// TIA Portal V15.1 export
// export: Created 2024-06-21T08:41:20.9813268Z, ExportSetting WithDefaults, DisplayName Totally Integrated Automation Portal, DisplayVersion V15.1 Update 5, DisplayName TIA Portal Openness, DisplayVersion V15.1 Update 5, DisplayName SINAMICS Startdrive Advanced, DisplayVersion V15.1, DisplayName G130, G150, S120, S150, SINAMICS MV, S210, DisplayVersion V15.1, DisplayName G110M, G120, G120C, G120D, G120P, DisplayVersion V15.1, DisplayName STEP 7 Professional, DisplayVersion V15.1 Update 5, DisplayName STEP 7 Safety, DisplayVersion V15.1, DisplayName WinCC Professional, DisplayVersion V15.1 Update 5, DisplayName SIMATIC Visualization Architect, DisplayVersion V15.1
FUNCTION_BLOCK "LVIDSMaster"   // FB1201, SCL
TITLE = LVIDSMaster
{ S7_Optimized_Access := 'FALSE' }
VERSION : 0.1
// stored: AutoNumber false, IsIECCheckEnabled false, SetENOAutomatically False, UDAEnableTagReadback false
   VAR_INPUT
      C_SubSystem { ExternalAccessible := 'False'; ExternalVisible := 'False'; ExternalWritable := 'False'} : Int;   // VDComm - Subsystem
      C_VDCommMasterRcvDB { ExternalAccessible := 'False'; ExternalVisible := 'False'; ExternalWritable := 'False'} : DB_ANY;   // VDComm - Master receive DB
      C_VDCommMasterSndDB { ExternalAccessible := 'False'; ExternalVisible := 'False'; ExternalWritable := 'False'} : DB_ANY;   // VDComm - Master send DB
      C_VDCommLocalRcvDB { ExternalAccessible := 'False'; ExternalVisible := 'False'; ExternalWritable := 'False'} : DB_ANY;   // VDComm - Local receive DB
      C_VDCommLocalSndDB { ExternalAccessible := 'False'; ExternalVisible := 'False'; ExternalWritable := 'False'} : DB_ANY;   // VDComm - Local send DB
      C_Plant { ExternalAccessible := 'False'; ExternalVisible := 'False'; ExternalWritable := 'False'} : Int;   // Plant ( VCG : 321, VCT : 461, VCCD : 861, VCQD : 862, VCLQ : 863, VCCH : 11 )
      C_IDType { ExternalAccessible := 'False'; ExternalVisible := 'False'; ExternalWritable := 'False'} : DWord;   // Identifier type (0 : Body tag, > 0 : Carrier tag Ex.: Carrier A-shop 162)
      I_OutOfUse { ExternalAccessible := 'False'; ExternalVisible := 'False'; ExternalWritable := 'False'} : Bool;   // Put out of use
      I_PartPres { ExternalAccessible := 'False'; ExternalVisible := 'False'; ExternalWritable := 'False'} : Bool;   // Cycle of tag data use active / Part is present in station
      I_TagID { ExternalAccessible := 'False'; ExternalVisible := 'False'; ExternalWritable := 'False'} : DWord;   // Tag identification ( to get VEM data )
      I_BodyID { ExternalAccessible := 'False'; ExternalVisible := 'False'; ExternalWritable := 'False'} : DWord;   // Body identification ( to get VEM data )
      I_CarrierID { ExternalAccessible := 'False'; ExternalVisible := 'False'; ExternalWritable := 'False'} : DWord;   // Carrier identification ( to get VEM data )
      I_MixNbr { ExternalAccessible := 'False'; ExternalVisible := 'False'; ExternalWritable := 'False'} : DWord;   // Mixnumber ( to get VEM data )
      I_PopID { ExternalAccessible := 'False'; ExternalVisible := 'False'; ExternalWritable := 'False'} : UDInt;   // Spare Data / PopID ( to get VEM data )
      I_PopIDSuffix { ExternalAccessible := 'False'; ExternalVisible := 'False'; ExternalWritable := 'False'} : Char;   // PopID suffix ( to get VEM data )
      I_PopType { ExternalAccessible := 'False'; ExternalVisible := 'False'; ExternalWritable := 'False'} : UDInt;   // Pop identifier ( to get VEM data )
      I_StartGetVEMData { ExternalAccessible := 'False'; ExternalVisible := 'False'; ExternalWritable := 'False'} : Bool;   // Get VEM data - Start on edge
      I_ResetAlarm { ExternalAccessible := 'False'; ExternalVisible := 'False'; ExternalWritable := 'False'} : Bool;   // Reset alarm
   END_VAR
   VAR_OUTPUT
      O_VEMDataValid { ExternalAccessible := 'False'; ExternalVisible := 'False'; ExternalWritable := 'False'} : Bool;   // VEM data is valid
      O_VEMDataNotValid { ExternalAccessible := 'False'; ExternalVisible := 'False'; ExternalWritable := 'False'} : Bool;   // VEM data is not valid
      O_GetVEMDataBusy { ExternalAccessible := 'False'; ExternalVisible := 'False'; ExternalWritable := 'False'} : Bool;   // Get VEM data - Busy
      O_Status { ExternalAccessible := 'False'; ExternalVisible := 'False'; ExternalWritable := 'False'} : Int;   // 0: no activity, 1: OK-Data valid, 2: Busy, -1..-32768: error code / 0: no activity, 1: OK-Get VEM data valid, 2: Busy, -1..-32768: error code
      O_Alarm { ExternalAccessible := 'False'; ExternalVisible := 'False'; ExternalWritable := 'False'} : Bool;   // Get VEM Data Alarm (Status < 0)
   END_VAR
   VAR_IN_OUT
      IO_VDComm : "VDComm";   // VD Comm / VD Comm - communication record
      IO_VIDS : "VIDS";   // VIDS - internal record
      IO_VEMData : "VEMData";   // VEM data - received
      IO_VEMDataChange : "VEMData";   // VEM data - to be changed
      IO_SpecificData : Array[0..7925] of Byte;   // Specific data received
      IO_Alarm : "Alarm";   // Alarm
      H_Master : "H_LVIDSMaster";   // Animation
      H_HMI : "H_HMI";   // Used for icon animation
   END_VAR
   VAR DB_SPECIFIC
      i { ExternalAccessible := 'False'; ExternalVisible := 'False'; ExternalWritable := 'False'} : Int;   // Index
      PartPres { ExternalAccessible := 'False'; ExternalVisible := 'False'; ExternalWritable := 'False'} : Bool;
      PartLostDlyTmrElapsed { ExternalAccessible := 'False'; ExternalVisible := 'False'; ExternalWritable := 'False'} : Bool;
      PartLostDlyTmrAct { ExternalAccessible := 'False'; ExternalVisible := 'False'; ExternalWritable := 'False'} : DInt;
      VEMDataChangeIoSerial { ExternalAccessible := 'False'; ExternalVisible := 'False'; ExternalWritable := 'False'} : Bool;
      VEMDataChangeHMISerial { ExternalAccessible := 'False'; ExternalVisible := 'False'; ExternalWritable := 'False'} : Array[0..255] of Byte;
      VEMDataChangeHMI { ExternalAccessible := 'False'; ExternalVisible := 'False'; ExternalWritable := 'False'; S7_SetPoint := 'True'} : "VEMData";
      VEMDataInitArray { ExternalAccessible := 'False'; ExternalVisible := 'False'; ExternalWritable := 'False'} : Array[0..255] of Byte;   // VEM data in serialized form
      VEMDataRcvArray { ExternalAccessible := 'False'; ExternalVisible := 'False'; ExternalWritable := 'False'} : Array[0..255] of Byte;   // VEM data in serialized form
      VEMDataRcv { ExternalAccessible := 'False'; ExternalVisible := 'False'; ExternalWritable := 'False'; S7_SetPoint := 'True'} : "VEMData";
      VEMDataSndArray { ExternalAccessible := 'False'; ExternalVisible := 'False'; ExternalWritable := 'False'} : Array[0..255] of Byte;
      SpecificData { ExternalAccessible := 'False'; ExternalVisible := 'False'; ExternalWritable := 'False'} : Array[0..7925] of Byte;
      VEMDataValid { ExternalAccessible := 'False'; ExternalVisible := 'False'; ExternalWritable := 'False'} : Bool;
      VEMDataNotValid { ExternalAccessible := 'False'; ExternalVisible := 'False'; ExternalWritable := 'False'} : Bool;
      CmdCodeSent { ExternalAccessible := 'False'; ExternalVisible := 'False'; ExternalWritable := 'False'} : DWord;   // Command code sent to VD
      CmdCodeRcvd { ExternalAccessible := 'False'; ExternalVisible := 'False'; ExternalWritable := 'False'} : DWord;   // Command code received from VD
      TagIDMem { ExternalAccessible := 'False'; ExternalVisible := 'False'; ExternalWritable := 'False'} : DWord;
      BodyIDMem { ExternalAccessible := 'False'; ExternalVisible := 'False'; ExternalWritable := 'False'} : DWord;
      CarrierIDMem { ExternalAccessible := 'False'; ExternalVisible := 'False'; ExternalWritable := 'False'} : DWord;
      MixNbrMem { ExternalAccessible := 'False'; ExternalVisible := 'False'; ExternalWritable := 'False'} : DWord;
      PopIDMem { ExternalAccessible := 'False'; ExternalVisible := 'False'; ExternalWritable := 'False'} : UDInt;   // Spare Data / PopID
      PopIDSuffixMem { ExternalAccessible := 'False'; ExternalVisible := 'False'; ExternalWritable := 'False'} : Char;   // PopID suffix
      PopTypeMem { ExternalAccessible := 'False'; ExternalVisible := 'False'; ExternalWritable := 'False'} : UDInt;   // Spare Data / Pop Identifier
      CarTypeVariant { ExternalAccessible := 'False'; ExternalVisible := 'False'; ExternalWritable := 'False'} : Int;   // Car type - Decoded from variant
      CarTypeBody { ExternalAccessible := 'False'; ExternalVisible := 'False'; ExternalWritable := 'False'} : Int;   // Car type - Decoded from bodytype matrix
      SteeringVariant { ExternalAccessible := 'False'; ExternalVisible := 'False'; ExternalWritable := 'False'} : Int;
      SteeringBody { ExternalAccessible := 'False'; ExternalVisible := 'False'; ExternalWritable := 'False'} : Int;
      CarTypeArray { ExternalAccessible := 'False'; ExternalVisible := 'False'; ExternalWritable := 'False'} : Array[1..3] of Int;
      DataValidSnd { ExternalAccessible := 'False'; ExternalVisible := 'False'; ExternalWritable := 'False'} : Bool;   // Data valid - Send
      DataRcvOk { ExternalAccessible := 'False'; ExternalVisible := 'False'; ExternalWritable := 'False'} : Bool;
      DataRcvNok { ExternalAccessible := 'False'; ExternalVisible := 'False'; ExternalWritable := 'False'} : Bool;
      DeserializePos { ExternalAccessible := 'False'; ExternalVisible := 'False'; ExternalWritable := 'False'} : DInt;
      SerializePos { ExternalAccessible := 'False'; ExternalVisible := 'False'; ExternalWritable := 'False'} : DInt;
      SequenceTotalOvertime { ExternalAccessible := 'False'; ExternalVisible := 'False'; ExternalWritable := 'False'} : Time;
      StartChangeVEMDataEdg { ExternalAccessible := 'False'; ExternalVisible := 'False'; ExternalWritable := 'False'} : Bool;   // Change VEM data - Start edge
      StartChangeVEMDataPls { ExternalAccessible := 'False'; ExternalVisible := 'False'; ExternalWritable := 'False'} : Bool;   // Change VEM data - Start pulse
      SeqOvTimeElapsed { ExternalAccessible := 'False'; ExternalVisible := 'False'; ExternalWritable := 'False'} : Bool;
      CodeBusy { ExternalAccessible := 'False'; ExternalVisible := 'False'; ExternalWritable := 'False'} : Int;
      RetVal { ExternalAccessible := 'False'; ExternalVisible := 'False'; ExternalWritable := 'False'} : Int;   // Return value
      GetVEMDataByRFIDBeginReqEdg { ExternalAccessible := 'False'; ExternalVisible := 'False'; ExternalWritable := 'False'} : Bool;
      GetVEMDataByTagReplBeginReqEdg { ExternalAccessible := 'False'; ExternalVisible := 'False'; ExternalWritable := 'False'} : Bool;
      DataValidRcvGetVEMDataByRFID { ExternalAccessible := 'False'; ExternalVisible := 'False'; ExternalWritable := 'False'} : Bool;
      GetVEMDataBeginReqEdg { ExternalAccessible := 'False'; ExternalVisible := 'False'; ExternalWritable := 'False'} : Bool;
      GetVEMDataByHMIBeginEdg { ExternalAccessible := 'False'; ExternalVisible := 'False'; ExternalWritable := 'False'} : Bool;
      GetVEMDataRcvOk { ExternalAccessible := 'False'; ExternalVisible := 'False'; ExternalWritable := 'False'} : Bool;
      ChangeDataReq { ExternalAccessible := 'False'; ExternalVisible := 'False'; ExternalWritable := 'False'} : Bool;
      ChangeDataReqEdg { ExternalAccessible := 'False'; ExternalVisible := 'False'; ExternalWritable := 'False'} : Bool;
      ChangeDataBeginReqEdg { ExternalAccessible := 'False'; ExternalVisible := 'False'; ExternalWritable := 'False'} : Bool;
      ChangeDataRcvOk { ExternalAccessible := 'False'; ExternalVisible := 'False'; ExternalWritable := 'False'} : Bool;
      GetNextIDBeginReqEdg { ExternalAccessible := 'False'; ExternalVisible := 'False'; ExternalWritable := 'False'} : Bool;
      GetNextIDRcvOk { ExternalAccessible := 'False'; ExternalVisible := 'False'; ExternalWritable := 'False'} : Bool;
      ReplaceTagReq { ExternalAccessible := 'False'; ExternalVisible := 'False'; ExternalWritable := 'False'} : Bool;
      ReplaceTagReqEdg { ExternalAccessible := 'False'; ExternalVisible := 'False'; ExternalWritable := 'False'} : Bool;
      ReplaceTagBeginReqEdg { ExternalAccessible := 'False'; ExternalVisible := 'False'; ExternalWritable := 'False'} : Bool;
      ReplaceTagRcvOk { ExternalAccessible := 'False'; ExternalVisible := 'False'; ExternalWritable := 'False'} : Bool;
      InitTagBeginReqEdg { ExternalAccessible := 'False'; ExternalVisible := 'False'; ExternalWritable := 'False'} : Bool;
      InitTagRcvOk { ExternalAccessible := 'False'; ExternalVisible := 'False'; ExternalWritable := 'False'} : Bool;
      GetSpecDataReq { ExternalAccessible := 'False'; ExternalVisible := 'False'; ExternalWritable := 'False'} : Bool;
      GetSpecDataReqEdg { ExternalAccessible := 'False'; ExternalVisible := 'False'; ExternalWritable := 'False'} : Bool;
      GetSpecDataBeginReqEdg { ExternalAccessible := 'False'; ExternalVisible := 'False'; ExternalWritable := 'False'} : Bool;
      GetSpecDataRcvOk { ExternalAccessible := 'False'; ExternalVisible := 'False'; ExternalWritable := 'False'} : Bool;
      PutSpecDataBeginReqEdg { ExternalAccessible := 'False'; ExternalVisible := 'False'; ExternalWritable := 'False'} : Bool;
      PutSpecDataRcvOk { ExternalAccessible := 'False'; ExternalVisible := 'False'; ExternalWritable := 'False'} : Bool;
      TrackBeginReqEdg { ExternalAccessible := 'False'; ExternalVisible := 'False'; ExternalWritable := 'False'} : Bool;   // Tracking - Begin request edge
      TrackingRcvOk { ExternalAccessible := 'False'; ExternalVisible := 'False'; ExternalWritable := 'False'} : Bool;
      CoupleBeginReqEdg { ExternalAccessible := 'False'; ExternalVisible := 'False'; ExternalWritable := 'False'} : Bool;
      CoupleRcvOk { ExternalAccessible := 'False'; ExternalVisible := 'False'; ExternalWritable := 'False'} : Bool;
      DecoupleBeginReqEdg { ExternalAccessible := 'False'; ExternalVisible := 'False'; ExternalWritable := 'False'} : Bool;
      DecoupleRcvOk { ExternalAccessible := 'False'; ExternalVisible := 'False'; ExternalWritable := 'False'} : Bool;
      ConfirmBeginReqEdg { ExternalAccessible := 'False'; ExternalVisible := 'False'; ExternalWritable := 'False'} : Bool;
      ConfirmationRcvOk { ExternalAccessible := 'False'; ExternalVisible := 'False'; ExternalWritable := 'False'} : Bool;
      NoFunctionBusy { ExternalAccessible := 'False'; ExternalVisible := 'False'; ExternalWritable := 'False'} : Bool;
      Busy { ExternalAccessible := 'False'; ExternalVisible := 'False'; ExternalWritable := 'False'} : Bool;
      BtnGetVEMTagIDEdge { ExternalAccessible := 'False'; ExternalVisible := 'False'; ExternalWritable := 'False'} : Bool;
      btnGetVEMDataByMixNbrEdg { ExternalAccessible := 'False'; ExternalVisible := 'False'; ExternalWritable := 'False'} : Bool;
      BtnGetVEMCarrierEdge { ExternalAccessible := 'False'; ExternalVisible := 'False'; ExternalWritable := 'False'} : Bool;
      ChangeDataNotValid { ExternalAccessible := 'False'; ExternalVisible := 'False'; ExternalWritable := 'False'} : Bool;
      MessageLength { ExternalAccessible := 'False'; ExternalVisible := 'False'; ExternalWritable := 'False'} : Word;   // Message Length
      SendToVD { ExternalAccessible := 'False'; ExternalVisible := 'False'; ExternalWritable := 'False'} : Bool;   // Send To PCS
      SendFinished { ExternalAccessible := 'False'; ExternalVisible := 'False'; ExternalWritable := 'False'} : Bool;   // Send Finished / Send data Finished
      RcvOkGetVEMDataCode { ExternalAccessible := 'False'; ExternalVisible := 'False'; ExternalWritable := 'False'} : Bool;
      RcvOkIdentification { ExternalAccessible := 'False'; ExternalVisible := 'False'; ExternalWritable := 'False'} : Bool;
      NewData { ExternalAccessible := 'False'; ExternalVisible := 'False'; ExternalWritable := 'False'} : Bool;   // New Data Is Present
      ResetNewData { ExternalAccessible := 'False'; ExternalVisible := 'False'; ExternalWritable := 'False'} : Bool;   // Reset Data Recevied
      CarrierIDDataReqOk { ExternalAccessible := 'False'; ExternalVisible := 'False'; ExternalWritable := 'False'} : Bool;
      ReqSendReport { ExternalAccessible := 'False'; ExternalVisible := 'False'; ExternalWritable := 'False'} : Bool;
      SendCmd { ExternalAccessible := 'False'; ExternalVisible := 'False'; ExternalWritable := 'False'} : Bool;   // External command send
      ResetAllRequests { ExternalAccessible := 'False'; ExternalVisible := 'False'; ExternalWritable := 'False'} : Bool;
      HMIGetVEMDataTagIDMem { ExternalAccessible := 'False'; ExternalVisible := 'False'; ExternalWritable := 'False'} : DInt;
      HMIGetVEMDataMixNbrMem { ExternalAccessible := 'False'; ExternalVisible := 'False'; ExternalWritable := 'False'} : DInt;
      HMIGetVEMDataCarrIdMem { ExternalAccessible := 'False'; ExternalVisible := 'False'; ExternalWritable := 'False'} : DInt;
      StartGetVEMDataEdg { ExternalAccessible := 'False'; ExternalVisible := 'False'; ExternalWritable := 'False'} : Bool;
      StartGetVEMDataPls { ExternalAccessible := 'False'; ExternalVisible := 'False'; ExternalWritable := 'False'} : Bool;
      Status { ExternalAccessible := 'False'; ExternalVisible := 'False'; ExternalWritable := 'False'} : Int;
      StatusMem { ExternalAccessible := 'False'; ExternalVisible := 'False'; ExternalWritable := 'False'} : Int;
      StepNbr { ExternalAccessible := 'False'; ExternalVisible := 'False'; ExternalWritable := 'False'} : Int;   // Active stepnumber
      Step0ExitPls { ExternalAccessible := 'False'; ExternalVisible := 'False'; ExternalWritable := 'False'} : Bool;   // Step 0 - Pulse created on exit
      Step50EntryEdg { ExternalAccessible := 'False'; ExternalVisible := 'False'; ExternalWritable := 'False'} : Bool;   // Step 50 - Edge created on entry
      Step50EntryPls { ExternalAccessible := 'False'; ExternalVisible := 'False'; ExternalWritable := 'False'} : Bool;   // Step 50 - Pulse created on entry
      Step50ExitEdg { ExternalAccessible := 'False'; ExternalVisible := 'False'; ExternalWritable := 'False'} : Bool;   // Step 50 - Edge created on exit
      Step50ExitPls { ExternalAccessible := 'False'; ExternalVisible := 'False'; ExternalWritable := 'False'} : Bool;   // Step 50 - Pulse created on exit
      Step100EntryEdg { ExternalAccessible := 'False'; ExternalVisible := 'False'; ExternalWritable := 'False'} : Bool;   // Step 100 - Edge created on entry
      Step100EntryPls { ExternalAccessible := 'False'; ExternalVisible := 'False'; ExternalWritable := 'False'} : Bool;   // Step 100 - Pulse created on entry
      Step100ExitEdg { ExternalAccessible := 'False'; ExternalVisible := 'False'; ExternalWritable := 'False'} : Bool;   // Step 100 - Edge created on exit
      Step100ExitPls { ExternalAccessible := 'False'; ExternalVisible := 'False'; ExternalWritable := 'False'} : Bool;   // Step 100 - Pulse created on exit
      Step200EntryEdg { ExternalAccessible := 'False'; ExternalVisible := 'False'; ExternalWritable := 'False'} : Bool;   // Step 200 - Edge created on entry
      Step200EntryPls { ExternalAccessible := 'False'; ExternalVisible := 'False'; ExternalWritable := 'False'} : Bool;   // Step 200 - Pulse created on entry
      Step200ExitEdg { ExternalAccessible := 'False'; ExternalVisible := 'False'; ExternalWritable := 'False'} : Bool;   // Step 200 - Edge created on exit
      Step200ExitPls { ExternalAccessible := 'False'; ExternalVisible := 'False'; ExternalWritable := 'False'} : Bool;   // Step 200 - Pulse created on exit
      Step300EntryEdg { ExternalAccessible := 'False'; ExternalVisible := 'False'; ExternalWritable := 'False'} : Bool;   // Step 300 - Edge created on entry
      Step300EntryPls { ExternalAccessible := 'False'; ExternalVisible := 'False'; ExternalWritable := 'False'} : Bool;   // Step 300 - Pulse created on entry
      Step300ExitEdg { ExternalAccessible := 'False'; ExternalVisible := 'False'; ExternalWritable := 'False'} : Bool;   // Step 300 - Edge created on exit
      Step300ExitPls { ExternalAccessible := 'False'; ExternalVisible := 'False'; ExternalWritable := 'False'} : Bool;   // Step 300 - Pulse created on exit
      Step400ExitEdg { ExternalAccessible := 'False'; ExternalVisible := 'False'; ExternalWritable := 'False'} : Bool;   // Step 400 - Edge created on exit
      Step400ExitPls { ExternalAccessible := 'False'; ExternalVisible := 'False'; ExternalWritable := 'False'} : Bool;   // Step 400 - Pulse created on exit
      Step0To50Cond { ExternalAccessible := 'False'; ExternalVisible := 'False'; ExternalWritable := 'False'} : Bool;   // Step 0 to 50 - Condition
      Step50To100Cond { ExternalAccessible := 'False'; ExternalVisible := 'False'; ExternalWritable := 'False'} : Bool;   // Step 0 to 100 - Condition
      Step50To200Cond { ExternalAccessible := 'False'; ExternalVisible := 'False'; ExternalWritable := 'False'} : Bool;   // Step 0 to 200 - Condition
      Step100To300Cond1 { ExternalAccessible := 'False'; ExternalVisible := 'False'; ExternalWritable := 'False'} : Bool;   // Step 100 to 300 - Condition 1
      Step100To300Cond2 { ExternalAccessible := 'False'; ExternalVisible := 'False'; ExternalWritable := 'False'} : Bool;   // Step 100 to 300 - Condition 2
      Step100To300Cond { ExternalAccessible := 'False'; ExternalVisible := 'False'; ExternalWritable := 'False'} : Bool;   // Step 100 to 300 - Condition
      Step200To300Cond { ExternalAccessible := 'False'; ExternalVisible := 'False'; ExternalWritable := 'False'} : Bool;   // Step 200 to 300 - Condition
      Step300To400Cond { ExternalAccessible := 'False'; ExternalVisible := 'False'; ExternalWritable := 'False'} : Bool;   // Step 300 to 400 - Condition
      Step300To400Cond1 { ExternalAccessible := 'False'; ExternalVisible := 'False'; ExternalWritable := 'False'} : Bool;   // Step 300 to 400 - Condition 1
      Step300To400Cond2 { ExternalAccessible := 'False'; ExternalVisible := 'False'; ExternalWritable := 'False'} : Bool;   // Step 300 to 400 - Condition 2
      Step400To0Cond { ExternalAccessible := 'False'; ExternalVisible := 'False'; ExternalWritable := 'False'} : Bool;   // Step 400 to 0 - Condition
      DataRcvOkGetSpecData { ExternalAccessible := 'False'; ExternalVisible := 'False'; ExternalWritable := 'False'} : Bool;
      VEMDataRcvOKCond1 { ExternalAccessible := 'False'; ExternalVisible := 'False'; ExternalWritable := 'False'} : Bool;
      VEMDataRcvOKCond2 { ExternalAccessible := 'False'; ExternalVisible := 'False'; ExternalWritable := 'False'} : Bool;
      VDCommLocalSndDB { ExternalAccessible := 'False'; ExternalVisible := 'False'; ExternalWritable := 'False'} : Int;   // Send DB / VD Comm - Local send DB number
      VDCommLocalRcvDB { ExternalAccessible := 'False'; ExternalVisible := 'False'; ExternalWritable := 'False'} : Int;   // Recv DB / VD Comm - Local receive DB number
      VD_Identification { ExternalAccessible := 'False'; ExternalVisible := 'False'; ExternalWritable := 'False'} : DWord;   // Identification from VD
      SpecDataLength_DW { ExternalAccessible := 'False'; ExternalVisible := 'False'; ExternalWritable := 'False'} : DWord;
      SpecDataLength_DInt { ExternalAccessible := 'False'; ExternalVisible := 'False'; ExternalWritable := 'False'} : DInt;
      TotalDataSentLength { ExternalAccessible := 'False'; ExternalVisible := 'False'; ExternalWritable := 'False'} : DInt;
      Cmd { ExternalAccessible := 'False'; ExternalVisible := 'False'; ExternalWritable := 'False'} : DWord;
      SeqOvTime { ExternalAccessible := 'False'; ExternalVisible := 'False'; ExternalWritable := 'False'} : Bool;
      OkBegin { ExternalAccessible := 'False'; ExternalVisible := 'False'; ExternalWritable := 'False'} : Bool;
      Step50TmrElapsed { ExternalAccessible := 'False'; ExternalVisible := 'False'; ExternalWritable := 'False'} : Bool;   // Step 50 - Step time elapsed
      Step50TmrAct { ExternalAccessible := 'False'; ExternalVisible := 'False'; ExternalWritable := 'False'} : DInt;   // Step 50 - Step time actual
      Step50TmrActMax { ExternalAccessible := 'False'; ExternalVisible := 'False'; ExternalWritable := 'False'} : DInt;   // Step 50 - Step time actual maximum
      Step100TmrElapsed { ExternalAccessible := 'False'; ExternalVisible := 'False'; ExternalWritable := 'False'} : Bool;   // Step 100 - Step time elapsed
      Step100TmrAct { ExternalAccessible := 'False'; ExternalVisible := 'False'; ExternalWritable := 'False'} : DInt;   // Step 100 - Step time actual
      Step100TmrActMax { ExternalAccessible := 'False'; ExternalVisible := 'False'; ExternalWritable := 'False'} : DInt;   // Step 100 - Step time actual maximum
      Step200TmrElapsed { ExternalAccessible := 'False'; ExternalVisible := 'False'; ExternalWritable := 'False'} : Bool;   // Step 200 - Step time elapsed
      Step200TmrAct { ExternalAccessible := 'False'; ExternalVisible := 'False'; ExternalWritable := 'False'} : DInt;   // Step 200 - Step time actual
      Step200TmrActMax { ExternalAccessible := 'False'; ExternalVisible := 'False'; ExternalWritable := 'False'} : DInt;   // Step 200 - Step time actual maximum
      Step300TmrElapsed { ExternalAccessible := 'False'; ExternalVisible := 'False'; ExternalWritable := 'False'} : Bool;   // Step 300 - Step time elapsed
      Step300TmrAct { ExternalAccessible := 'False'; ExternalVisible := 'False'; ExternalWritable := 'False'} : DInt;   // Step 300 - Step time actual
      Step300TmrActMax { ExternalAccessible := 'False'; ExternalVisible := 'False'; ExternalWritable := 'False'} : DInt;   // Step 300 - Step time actual maximum
      Step400TmrElapsed { ExternalAccessible := 'False'; ExternalVisible := 'False'; ExternalWritable := 'False'} : Bool;   // Step 400 - Step time elapsed
      Step400TmrAct { ExternalAccessible := 'False'; ExternalVisible := 'False'; ExternalWritable := 'False'} : DInt;   // Step 400 - Step time actual
      Step400TmrActMax { ExternalAccessible := 'False'; ExternalVisible := 'False'; ExternalWritable := 'False'} : DInt;   // Step 400 - Step time actual maximum
      EmptyByte { ExternalAccessible := 'False'; ExternalVisible := 'False'; ExternalWritable := 'False'} : Byte;
      PartLostEdg { ExternalAccessible := 'False'; ExternalVisible := 'False'; ExternalWritable := 'False'} : Bool;   // Part lost edge
      PartLostPls { ExternalAccessible := 'False'; ExternalVisible := 'False'; ExternalWritable := 'False'} : Bool;   // Part lost pulse
      PutVemDataTotalLength { ExternalAccessible := 'False'; ExternalVisible := 'False'; ExternalWritable := 'False'} : DInt;
      DataValidRcv { ExternalAccessible := 'False'; ExternalVisible := 'False'; ExternalWritable := 'False'} : Bool;
      BusyGetVEMData { ExternalAccessible := 'False'; ExternalVisible := 'False'; ExternalWritable := 'False'} : Bool;
      Alarm { ExternalAccessible := 'False'; ExternalVisible := 'False'; ExternalWritable := 'False'} : Bool;   // Alarm
      msgPartPresVisible { ExternalAccessible := 'False'; ExternalVisible := 'False'; ExternalWritable := 'False'} : Word;   // HMI - Message animation - Part present - Visible
      msgPartPresAnim { ExternalAccessible := 'False'; ExternalVisible := 'False'; ExternalWritable := 'False'} : Word;   // HMI - Message animation - Part present - Summary
      msgPartNotPresVisible { ExternalAccessible := 'False'; ExternalVisible := 'False'; ExternalWritable := 'False'} : Word;   // HMI - Message animation - Part not present - Visible
      msgPartNotPresAnim { ExternalAccessible := 'False'; ExternalVisible := 'False'; ExternalWritable := 'False'} : Word;   // HMI - Message animation - Part not present - Summary
      IconColour { ExternalAccessible := 'False'; ExternalVisible := 'False'; ExternalWritable := 'False'} : Word;   // Icon colour
      SPACE { ExternalAccessible := 'False'; ExternalVisible := 'False'; ExternalWritable := 'False'} : Char := ' ';
   END_VAR
   VAR
      _Step50Tmr { ExternalAccessible := 'False'; ExternalVisible := 'False'; ExternalWritable := 'False'; S7_SetPoint := 'True'} : "LTimer";   // Step 50 - Timer
      _Step100Tmr { ExternalAccessible := 'False'; ExternalVisible := 'False'; ExternalWritable := 'False'; S7_SetPoint := 'True'} : "LTimer";   // Step 100 - Timer
      _Step200Tmr { ExternalAccessible := 'False'; ExternalVisible := 'False'; ExternalWritable := 'False'; S7_SetPoint := 'True'} : "LTimer";   // Step 200 - Timer
      _Step300Tmr { ExternalAccessible := 'False'; ExternalVisible := 'False'; ExternalWritable := 'False'; S7_SetPoint := 'True'} : "LTimer";   // Step 300 - Timer
      "_LVDComSubSystemS7-1500" { ExternalAccessible := 'False'; ExternalVisible := 'False'; ExternalWritable := 'False'; S7_SetPoint := 'True'} : "LVDComSubSystemS7-1500";
      _PartLostDlyTmr { ExternalAccessible := 'False'; ExternalVisible := 'False'; ExternalWritable := 'False'; S7_SetPoint := 'True'} : "LTimer";   // Part present lost delay timer
   END_VAR
   VAR_TEMP
      ptrIO_VEMData : Any;   // Pointer to received VEM data / Pointer to IO_VEM data
      ptrIO_VEMDataStruct AT ptrIO_VEMData : Struct   // Pointer to IO_VEM data - Structure
         ID : Byte;
         DataType : Byte;
         ReplicationFactor : Word;
         DbNbr : Word;
         CrossAreaPointer : DWord;
      END_STRUCT;
      ptrIO_VEMDataChange : Any;   // Pointer to received VEM data / Pointer to IO_VEM data Change
      ptrIO_VEMDataChangeStruct AT ptrIO_VEMDataChange : Struct   // Pointer to IO_VEM data Change - Structure
         ID : Byte;
         DataType : Byte;
         ReplicationFactor : Word;
         DbNbr : Word;
         CrossAreaPointer : DWord;
      END_STRUCT;
      ptrIO_SpecData : Any;   // Pointer to received VEM data / Pointer to IO_Specific data
      ptrIO_SpecDataStruct AT ptrIO_SpecData : Struct   // Pointer to IO_Specific data - Structure
         ID : Byte;
         DataType : Byte;
         ReplicationFactor : Word;
         DbNbr : Word;
         CrossAreaPointer : DWord;
      END_STRUCT;
      ptrVEMDataVDCommLocalRcv : Any;   // Pointer to received VEM data / Pointer to VEM data in VD local receive DB
      ptrVEMDataVDCommLocalRcvStruct AT ptrVEMDataVDCommLocalRcv : Struct   // Pointer to VEM data in VD local receive DB - Structure
         ID : Byte;
         DataType : Byte;
         ReplicationFactor : Word;
         DbNbr : Word;
         CrossAreaPointer : DWord;
      END_STRUCT;
      ptrVEMDataVDCommLocalSnd : Any;   // Pointer to VEM and specific data to be sent / Pointer to VEM data in VD local send DB
      ptrVEMDataVDCommLocalSndStruct AT ptrVEMDataVDCommLocalSnd : Struct   // Pointer to VEM data in VD local send DB - Structure
         ID : Byte;
         DataType : Byte;
         ReplicationFactor : Word;
         DbNbr : Word;
         CrossAreaPointer : DWord;
      END_STRUCT;
      ptrSpecDataVDCommLocalRcv : Any;   // Pointer to received specific data / Pointer to Specific data in VD local receive DB
      ptrSpecDataVDCommLocalRcvStruct AT ptrSpecDataVDCommLocalRcv : Struct   // Pointer to Specific data in VD local receive DB - Structure
         ID : Byte;
         DataType : Byte;
         ReplicationFactor : Word;
         DbNbr : Word;
         CrossAreaPointer : DWord;
      END_STRUCT;
      ptrSpecDataVDCommLocalSnd : Any;   // Pointer to VEM and specific data to be sent / Pointer to Specific data in VD local send DB
      ptrSpecDataVDCommLocalSndStruct AT ptrSpecDataVDCommLocalSnd : Struct   // Pointer to Specific data in VD local send DB - Structure
         ID : Byte;
         DataType : Byte;
         ReplicationFactor : Word;
         DbNbr : Word;
         CrossAreaPointer : DWord;
      END_STRUCT;
   END_VAR
   VAR CONSTANT
      SECTION_OUTPUTS : Bool := TRUE;   // Section - Outputs
      SECTION_HMI : Bool := TRUE;   // Section - HMI
      PART_LOST_DLY : DInt := 1000;
      VEM_DATA_OFFSET : DWord;
      SPEC_DATA_OFFSET : DWord := 16#100;
      VDCOM_DATA_OFFSET : DWord := 10;
      VDCOM_VEM_DATA_OFFSET : DWord := 10;
      VDCOM_SPEC_DATA_OFFSET : DWord := 266;
      DATA_TYPE_BYTE : Byte := 16#02;
      AREA_IDENTIFIER : DWord := 16#84000000;
      POINTER_SYNTAX_ID : Byte := 16#10;
      ON : Word := 16#0001;
      OFF : Word := 16#0000;
      DATA_SND_TIME_MAX : Time := T#10S;
      DATA_RCV_TIME_MAX : Time := T#15S;
      STAT_CODE_BUSY : Int := 2;   // Status code - job busy
      STAT_CODE_SUCCESS : Int := 1;   // Status code - job successful
      STAT_CODE_SND_FINISH_NOK : Int := -3;   // Status code - No Send finished
      STAT_CODE_START_WITHOUT_ID : Int := -4;   // Status code - ID not valid or missing
      STAT_CODE_RCV_DATA_NOK : Int := -5;   // Status code - Received data is NOK
      STAT_CODE_RCV_NEW_DATA_OVTIME : Int := -9;   // Status code - New Data Received Overtime
      CMD_GET_VEM_DATA : DWord := 1002;
      SPECIFIC_DATA_LENGTH_MAX : DInt := 7026;
      STATUS_001 : Int := 1;   // Status - 001 : Success
      STATUS_MINUS_003 : Int := -3;   // Status - 003 : Error sending message to virtual device
      STATUS_MINUS_006 : Int := -6;   // Status - 006 : Error ID not valid or missing
      STATUS_MINUS_001 : Int := -1;   // Status - 001 :
      STATUS_MINUS_005 : Int := -5;   // Status -009 : Error no response received from virtual device
      STATUS_MINUS_009 : Int := -9;   // Status -009 : Error no response received from virtual device
      VISIBLE : Word := 16#0001;   // Enable
      ENABLE : Word := 16#0002;   // Visible
      COLOUR_DEFAULT : Word := 16#0000;   // Colour - Default
      COLOUR_RED : Word := 16#0010;   // Colour - Red
      COLOUR_GREEN : Word := 16#0020;   // Colour - Green
      COLOUR_BLUE : Word := 16#0040;   // Colour - Blue
      COLOUR_WHITE : Word := 16#0080;   // Colour - White
      COLOUR_BLUE_FLASH : Word := 16#0400;   // Colour - Blue flash
   END_VAR
BEGIN
   (******************************************************************************
    Changelog

       17W24D4 10:00H PMo
       - Section outputs is now true

       17W23D5 17:00H PMo
       - Conversion from FBD TO SCL

       18W3D5 : AHE
       - Confirm.ok.begin will not clear VEM data

    19W12D4 : WDL
       - Decoding of BodyTypeMatrix removed

    List OF authors

       Company : Volvo Cars Gent
       Name    : Patrick Moreau (PMo)
       E-mail  : patrick.moreau@volvocars.com
       Tel.    : +32 9 2503165

    Description

       This module is part OF the VIDS suite AND is the principal module TO be
       integrated FOR RFID, Track, Confirm AND other submodules.
       Its main purpose is TO communicate with the production servers via virtual
       device AND retrieve VEM data OR specific data 

    ******************************************************************************)

   (******************************************************************************)
   (* Create pointers                                                            *)
   (******************************************************************************)

   //Copy pointers
   #ptrIO_VEMData := #IO_VEMData;
   #ptrIO_VEMDataChange := #IO_VEMDataChange;
   #ptrIO_SpecData := #IO_SpecificData;

   //Create pointer to VEMData in VDComm local receive DB
   #ptrVEMDataVDCommLocalRcvStruct.ID := #POINTER_SYNTAX_ID;
   #ptrVEMDataVDCommLocalRcvStruct.DataType := #DATA_TYPE_BYTE;
   #ptrVEMDataVDCommLocalRcvStruct.ReplicationFactor := 256;
   #ptrVEMDataVDCommLocalRcvStruct.DbNbr := UINT_TO_WORD(DB_ANY_TO_UINT(#C_VDCommLocalRcvDB));
   #ptrVEMDataVDCommLocalRcvStruct.CrossAreaPointer := SHL(IN := #VDCOM_VEM_DATA_OFFSET, N := 3) OR #AREA_IDENTIFIER; //Offset 10

   //Create pointer to Specific data in VDComm local receive DB
   #ptrSpecDataVDCommLocalRcvStruct.ID := #POINTER_SYNTAX_ID;
   #ptrSpecDataVDCommLocalRcvStruct.DataType := #DATA_TYPE_BYTE;
   #ptrSpecDataVDCommLocalRcvStruct.ReplicationFactor := 7026;
   #ptrSpecDataVDCommLocalRcvStruct.DbNbr := UINT_TO_WORD(DB_ANY_TO_UINT(#C_VDCommLocalRcvDB));
   #ptrSpecDataVDCommLocalRcvStruct.CrossAreaPointer := SHL(IN := #VDCOM_SPEC_DATA_OFFSET, N := 3) OR #AREA_IDENTIFIER; //Offset 266

   //Create pointer to VEMData in VDComm local send DB
   #ptrVEMDataVDCommLocalSndStruct.ID := #POINTER_SYNTAX_ID;
   #ptrVEMDataVDCommLocalSndStruct.DataType := #DATA_TYPE_BYTE;
   #ptrVEMDataVDCommLocalSndStruct.ReplicationFactor := 256;
   #ptrVEMDataVDCommLocalSndStruct.DbNbr := UINT_TO_WORD(DB_ANY_TO_UINT(#C_VDCommLocalSndDB));
   #ptrVEMDataVDCommLocalSndStruct.CrossAreaPointer := SHL(IN := #VDCOM_VEM_DATA_OFFSET, N := 3) OR #AREA_IDENTIFIER; //Offset 10

   //Create pointer to Specific data in VDComm local send DB
   #ptrSpecDataVDCommLocalSndStruct.ID := #POINTER_SYNTAX_ID;
   #ptrSpecDataVDCommLocalSndStruct.DataType := #DATA_TYPE_BYTE;
   #ptrSpecDataVDCommLocalSndStruct.ReplicationFactor := 2048;
   #ptrSpecDataVDCommLocalSndStruct.DbNbr := UINT_TO_WORD(DB_ANY_TO_UINT(#C_VDCommLocalSndDB));
   #ptrSpecDataVDCommLocalSndStruct.CrossAreaPointer := SHL(IN := #VDCOM_SPEC_DATA_OFFSET, N := 3) OR #AREA_IDENTIFIER; //Offset 266

   (******************************************************************************)
   (* Inputs                                                                     *)
   (******************************************************************************)

   #_PartLostDlyTmr(I_StartTimer:=#PartPres AND NOT #I_PartPres,
                 I_HoldTimer:=FALSE,
                 I_MaxTimerValue:=#PART_LOST_DLY,
                 O_TimerResult=>#PartLostDlyTmrElapsed,
                 O_TimerValue=>#PartLostDlyTmrAct);

   #PartPres := #I_PartPres OR #PartPres AND NOT #PartLostDlyTmrElapsed;

   (******************************************************************************)
   (* Create pulses                                                              *)
   (******************************************************************************)

   //Get VEM Data - Create start pulse
   #StartGetVEMDataPls := #I_StartGetVEMData AND NOT #StartGetVEMDataEdg;
   #StartGetVEMDataEdg := #I_StartGetVEMData;

   //Create pulse on part lost
   #PartLostPls := NOT #IO_VIDS.PartPres AND #PartLostEdg;
   #PartLostEdg := #IO_VIDS.PartPres;

   (******************************************************************************)
   (* Initialize all                                                             *)
   (******************************************************************************)

   IF #PartLostPls THEN

       #RetVal := FILL(BVAL := #EmptyByte, BLK => #VEMDataInitArray);  //Create init array
       #StepNbr := 0;                                                  //Reset sequence
       #VEMDataValid := FALSE;                                 //Reset VEM data valid
       #VEMDataNotValid := FALSE;                              //Reset VEM data not valid
       #Status := 0;                                                   //Reset status

       //Initialize IO_VIDS.VEMData
       #DeserializePos := 0;
       #RetVal := Deserialize(SRC_ARRAY := #VEMDataInitArray, DEST_VARIABLE => #IO_VIDS.VEMData, POS := #DeserializePos);
       #RetVal := FILL(BVAL := #SPACE, BLK => #IO_VIDS.VEMData.UserID);
       #RetVal := FILL(BVAL := #SPACE, BLK => #IO_VIDS.VEMData.Variant);
       #RetVal := FILL(BVAL := #SPACE, BLK => #IO_VIDS.VEMData.VinNumber);
       #RetVal := FILL(BVAL := #SPACE, BLK => #IO_VIDS.VEMData.PopIDSuffix);

       //Initialize IO_VIDS.Specific data
       #RetVal := FILL(BVAL := #EmptyByte, BLK => #IO_VIDS.SpecificDataInit);

       //Initialize IO_VEMData
       #DeserializePos := 0;
       #RetVal:=Deserialize(SRC_ARRAY := #VEMDataInitArray, DEST_VARIABLE => #IO_VEMData, POS := #DeserializePos);
       #RetVal := FILL(BVAL := #SPACE, BLK => #IO_VEMData.UserID);
       #RetVal := FILL(BVAL := #SPACE, BLK => #IO_VEMData.Variant);
       #RetVal := FILL(BVAL := #SPACE, BLK => #IO_VEMData.VinNumber);
       #RetVal := FILL(BVAL := #SPACE, BLK => #IO_VEMData.PopIDSuffix);

       //Initialize IO_Specific data
       #RetVal := FILL(BVAL := #EmptyByte, BLK => #IO_SpecificData);

       //Initialize IO_VEMDataChange
       #DeserializePos := 0;
       #RetVal := Deserialize(SRC_ARRAY := #VEMDataInitArray, DEST_VARIABLE => #IO_VEMDataChange, POS := #DeserializePos);
       #RetVal := FILL(BVAL := #SPACE, BLK => #IO_VEMDataChange.UserID);
       #RetVal := FILL(BVAL := #SPACE, BLK => #IO_VEMDataChange.Variant);
       #RetVal := FILL(BVAL := #SPACE, BLK => #IO_VEMDataChange.VinNumber);
       #RetVal := FILL(BVAL := #SPACE, BLK => #IO_VEMDataChange.PopIDSuffix);

       //Reset signals
       #IO_VIDS.GetVEMData.BeginReqMem := FALSE;
       #IO_VIDS.GetVEMData.Running := FALSE;

       #IO_VIDS.ChangeData.BeginReqMem := FALSE;
       #IO_VIDS.ChangeData.Running := FALSE;

       #IO_VIDS.InitTag.BeginReqMem := FALSE;
       #IO_VIDS.InitTag.Running := FALSE;

       #IO_VIDS.GetVEMDataByRFID.BeginReqMem := FALSE;
       #IO_VIDS.GetVEMDataByRFID.Running := FALSE;

       #IO_VIDS.ReplaceTag.BeginReqMem := FALSE;
       #IO_VIDS.ReplaceTag.Running := FALSE;

       #IO_VIDS.Confirm.BeginReqMem := FALSE;
       #IO_VIDS.Confirm.Running := FALSE;

       #IO_VIDS.Track.BeginReqMem := FALSE;
       #IO_VIDS.Track.Running := FALSE;

       #IO_VIDS.Couple.BeginReqMem := FALSE;
       #IO_VIDS.Couple.Running := FALSE;

       #IO_VIDS.DeCouple.BeginReqMem := FALSE;
       #IO_VIDS.DeCouple.Running := FALSE;

       #IO_VIDS.GetNextID.BeginReqMem := FALSE;
       #IO_VIDS.GetNextID.Running := FALSE;

       #IO_VIDS.GetSpecData.BeginReqMem := FALSE;
       #IO_VIDS.GetSpecData.Running := FALSE;

       #IO_VIDS.PutSpecData.BeginReqMem := FALSE;
       #IO_VIDS.PutSpecData.Running := FALSE;

   END_IF;

   //Running summary
   #Busy :=
   #IO_VIDS.GetVEMData.Running OR
   #IO_VIDS.ChangeData.Running OR
   #IO_VIDS.InitTag.Running OR
   #IO_VIDS.GetVEMDataByRFID.Running OR
   #IO_VIDS.ReplaceTag.Running OR
   #IO_VIDS.Track.Running OR
   #IO_VIDS.Confirm.Running OR
   #IO_VIDS.Couple.Running OR
   #IO_VIDS.DeCouple.Running OR
   #IO_VIDS.GetNextID.Running OR
   #IO_VIDS.GetSpecData.Running OR
   #IO_VIDS.PutSpecData.Running;

   (******************************************************************************)
   (* Get VEM data                                                               *)
   (******************************************************************************)

   //Get VEM Data - Begin request
   #IO_VIDS.GetVEMData.BeginReq := #StartGetVEMDataPls;

   //Get VEM data - Memorize parameters
   IF #IO_VIDS.GetVEMData.BeginReq THEN
       #TagIDMem := #I_TagID;
       #BodyIDMem := #I_BodyID;
       #CarrierIDMem := #I_CarrierID;
       #MixNbrMem := #I_MixNbr;
       #PopIDMem := #I_PopID;
       #PopIDSuffixMem := #I_PopIDSuffix;
       #PopTypeMem := #I_PopType;

   END_IF;

   //Get VEM data - Initialize parameters
   IF #IO_VIDS.GetVEMData.OkBegin THEN

       #IO_VIDS.VEMData.CommandCode := #CMD_GET_VEM_DATA;
       #IO_VIDS.VEMData.Identification := #TagIDMem;
       #IO_VIDS.VEMData.BodyID := #BodyIDMem;
       #IO_VIDS.VEMData.CarrierID := #CarrierIDMem;
       #IO_VIDS.VEMData.MixNumber := #MixNbrMem;
       #IO_VIDS.VEMData.IdType := #C_IDType;
       #IO_VIDS.VEMData.PopID := #PopIDMem;
       #IO_VIDS.VEMData.PopIDSuffix := #PopIDSuffixMem;
       #IO_VIDS.VEMData.PopType := #PopTypeMem;
   END_IF;

   //Get VEM data - Begin
   #IO_VIDS.GetVEMData.Begin := #IO_VIDS.GetVEMData.OkBegin;

   //Get VEM Data - Busy
   #BusyGetVEMData := #IO_VIDS.GetVEMData.Running;

   (******************************************************************************)
   (* Memorize begin request                                                     *)
   (******************************************************************************)

   //Get VEM Data - Memorize begin request
   IF #IO_VIDS.GetVEMData.BeginReq AND NOT #GetVEMDataBeginReqEdg THEN
       #IO_VIDS.GetVEMData.BeginReqMem := TRUE;
   END_IF;
   #GetVEMDataBeginReqEdg := #IO_VIDS.GetVEMData.BeginReq;

   //Change VEM Data - Memorize begin request
   IF #IO_VIDS.ChangeData.BeginReq AND NOT #ChangeDataBeginReqEdg THEN
       #IO_VIDS.ChangeData.BeginReqMem := TRUE;
   END_IF;
   #ChangeDataBeginReqEdg := #IO_VIDS.ChangeData.BeginReq;

   //Init tag - Memorize begin request
   IF #IO_VIDS.InitTag.BeginReq AND NOT #InitTagBeginReqEdg THEN
       #IO_VIDS.InitTag.BeginReqMem := TRUE;
   END_IF;
   #InitTagBeginReqEdg := #IO_VIDS.InitTag.BeginReq;

   //Get VEM Data by RFID - Memorize begin request
   IF #IO_VIDS.GetVEMDataByRFID.BeginReq AND NOT #GetVEMDataByRFIDBeginReqEdg THEN
       #IO_VIDS.GetVEMDataByRFID.BeginReqMem := TRUE;
   END_IF;
   #GetVEMDataByRFIDBeginReqEdg := #IO_VIDS.GetVEMDataByRFID.BeginReq;

   //Replace tag - Memorize begin request
   IF #IO_VIDS.ReplaceTag.BeginReq AND NOT #ReplaceTagBeginReqEdg THEN
       #IO_VIDS.ReplaceTag.BeginReqMem := TRUE;
   END_IF;
   #ReplaceTagBeginReqEdg := #IO_VIDS.ReplaceTag.BeginReq;

   //Track - Memorize begin request
   IF #IO_VIDS.Track.BeginReq AND NOT #TrackBeginReqEdg THEN
       #IO_VIDS.Track.BeginReqMem := TRUE;
   END_IF;
   #TrackBeginReqEdg := #IO_VIDS.Track.BeginReq;

   //Confirm - Memorize begin request
   IF #IO_VIDS.Confirm.BeginReq AND NOT #ConfirmBeginReqEdg THEN
       #IO_VIDS.Confirm.BeginReqMem := TRUE;
   END_IF;
   #ConfirmBeginReqEdg := #IO_VIDS.Confirm.BeginReq;

   //Couple - Memorize begin request
   IF #IO_VIDS.Couple.BeginReq AND NOT #CoupleBeginReqEdg THEN
       #IO_VIDS.Couple.BeginReqMem := TRUE;
   END_IF;
   #CoupleBeginReqEdg := #IO_VIDS.Couple.BeginReq;

   //Decouple - Memorize begin request
   IF #IO_VIDS.DeCouple.BeginReq AND NOT #DecoupleBeginReqEdg THEN
       #IO_VIDS.DeCouple.BeginReqMem := TRUE;
   END_IF;
   #DecoupleBeginReqEdg := #IO_VIDS.DeCouple.BeginReq;

   //Get next ID - Memorize begin request
   IF #IO_VIDS.GetNextID.BeginReq AND NOT #GetNextIDBeginReqEdg THEN
       #IO_VIDS.GetNextID.BeginReqMem := TRUE;
   END_IF;
   #GetNextIDBeginReqEdg := #IO_VIDS.GetNextID.BeginReq;

   //Get Specific data - Memorize begin request
   IF #IO_VIDS.GetSpecData.BeginReq AND NOT #GetSpecDataBeginReqEdg THEN
       #IO_VIDS.GetSpecData.BeginReqMem := TRUE;
   END_IF;
   #GetSpecDataBeginReqEdg := #IO_VIDS.GetSpecData.BeginReq;

   //Put specific data - Memorize begin request
   IF #IO_VIDS.PutSpecData.BeginReq AND NOT #PutSpecDataBeginReqEdg THEN
       #IO_VIDS.PutSpecData.BeginReqMem := TRUE;
   END_IF;
   #PutSpecDataBeginReqEdg := #IO_VIDS.PutSpecData.BeginReq;

   (******************************************************************************)
   (* Running                                                                    *)
   (******************************************************************************)

   IF #IO_VIDS.GetVEMData.OkBegin AND #IO_VIDS.GetVEMData.Begin THEN
       #IO_VIDS.GetVEMData.Running := TRUE;
   ELSIF #IO_VIDS.ChangeData.OkBegin AND #IO_VIDS.ChangeData.Begin THEN
       #IO_VIDS.ChangeData.Running := TRUE;
   ELSIF #IO_VIDS.InitTag.OkBegin AND #IO_VIDS.InitTag.Begin THEN
       #IO_VIDS.InitTag.Running := TRUE;
   ELSIF #IO_VIDS.GetVEMDataByRFID.OkBegin AND #IO_VIDS.GetVEMDataByRFID.Begin THEN
       #IO_VIDS.GetVEMDataByRFID.Running := TRUE;
   ELSIF #IO_VIDS.ReplaceTag.OkBegin AND #IO_VIDS.ReplaceTag.Begin THEN
       #IO_VIDS.ReplaceTag.Running := TRUE;
   ELSIF #IO_VIDS.Track.OkBegin AND #IO_VIDS.Track.Begin THEN
       #IO_VIDS.Track.Running := TRUE;
   ELSIF #IO_VIDS.Confirm.OkBegin AND #IO_VIDS.Confirm.Begin THEN
       #IO_VIDS.Confirm.Running := TRUE;
   ELSIF #IO_VIDS.Couple.OkBegin AND #IO_VIDS.Couple.Begin THEN
       #IO_VIDS.Couple.Running := TRUE;
   ELSIF #IO_VIDS.DeCouple.OkBegin AND #IO_VIDS.DeCouple.Begin THEN
       #IO_VIDS.DeCouple.Running := TRUE;
   ELSIF #IO_VIDS.GetNextID.OkBegin AND #IO_VIDS.GetNextID.Begin THEN
       #IO_VIDS.GetNextID.Running := TRUE;
   ELSIF #IO_VIDS.GetSpecData.OkBegin AND #IO_VIDS.GetSpecData.Begin THEN
       #IO_VIDS.GetSpecData.Running := TRUE;
   ELSIF #IO_VIDS.PutSpecData.OkBegin AND #IO_VIDS.PutSpecData.Begin THEN
       #IO_VIDS.PutSpecData.Running := TRUE;
   END_IF;

   (******************************************************************************)
   (* Update status                                                              *)
   (******************************************************************************)

   IF #StepNbr > 0 THEN
       IF #IO_VIDS.GetVEMData.Running THEN
           #IO_VIDS.GetVEMData.Status := #Status;
       ELSIF #IO_VIDS.ChangeData.Running THEN
           #IO_VIDS.ChangeData.Status := #Status;
       ELSIF #IO_VIDS.InitTag.Running THEN
           #IO_VIDS.InitTag.Status := #Status;
       ELSIF #IO_VIDS.GetVEMDataByRFID.Running THEN
           #IO_VIDS.GetVEMDataByRFID.Status := #Status;
       ELSIF #IO_VIDS.ReplaceTag.Running THEN
           #IO_VIDS.ReplaceTag.Status := #Status;
       ELSIF #IO_VIDS.Track.Running THEN
           #IO_VIDS.Track.Status := #Status;
       ELSIF #IO_VIDS.Confirm.Running THEN
           #IO_VIDS.Confirm.Status := #Status;
       ELSIF #IO_VIDS.Couple.Running THEN
           #IO_VIDS.Couple.Status := #Status;
       ELSIF #IO_VIDS.DeCouple.Running THEN
           #IO_VIDS.DeCouple.Status := #Status;
       ELSIF #IO_VIDS.GetNextID.Running THEN
           #IO_VIDS.GetNextID.Status := #Status;
       ELSIF #IO_VIDS.GetSpecData.Running THEN
           #IO_VIDS.GetSpecData.Status := #Status;
       ELSIF #IO_VIDS.PutSpecData.Running THEN
           #IO_VIDS.PutSpecData.Status := #Status;
       END_IF;
   END_IF;

   (******************************************************************************)
   (* Step 0                                                                     *)
   (******************************************************************************)

   //Step 0 On Active - Reset locked
   //IF #StepNbr = 0 THEN

   //END_IF;

   (******************************************************************************)
   (* Step 0 TO 50                                                               *)
   (******************************************************************************)

   //Step 0 to 50
   IF #Step0To50Cond THEN
       #StepNbr := 50;
       #Step50EntryPls := TRUE;
   ELSE
       #Step50EntryPls := FALSE;
   END_IF;

   //Step 0 to 50 - Condition
   #Step0To50Cond :=
   #StepNbr = 0 AND (
   #IO_VIDS.GetVEMData.BeginReqMem OR
   #IO_VIDS.ChangeData.BeginReqMem OR
   #IO_VIDS.InitTag.BeginReqMem OR
   #IO_VIDS.GetVEMDataByRFID.BeginReqMem OR
   #IO_VIDS.ReplaceTag.BeginReqMem OR
   #IO_VIDS.Track.BeginReqMem OR
   #IO_VIDS.Confirm.BeginReqMem OR
   #IO_VIDS.Couple.BeginReqMem OR
   #IO_VIDS.DeCouple.BeginReqMem OR
   #IO_VIDS.GetNextID.BeginReqMem OR
   #IO_VIDS.GetSpecData.BeginReqMem OR
   #IO_VIDS.PutSpecData.BeginReqMem);

   (******************************************************************************)
   (* Step 50                                                                    *)
   (******************************************************************************)

   //Step 50 On Entry
   IF #Step50EntryPls THEN

       //Ok Begin
       IF #IO_VIDS.GetVEMData.BeginReqMem  THEN
           #IO_VIDS.GetVEMData.OkBegin := TRUE;
           #IO_VIDS.GetVEMData.BeginReqMem := FALSE;
       ELSIF #IO_VIDS.ChangeData.BeginReqMem  THEN
           #IO_VIDS.ChangeData.OkBegin := TRUE;
           #IO_VIDS.ChangeData.BeginReqMem := FALSE;
       ELSIF #IO_VIDS.InitTag.BeginReqMem  THEN
           #IO_VIDS.InitTag.OkBegin := TRUE;
           #IO_VIDS.InitTag.BeginReqMem := FALSE;
       ELSIF #IO_VIDS.GetVEMDataByRFID.BeginReqMem  THEN
           #IO_VIDS.GetVEMDataByRFID.OkBegin := TRUE;
           #IO_VIDS.GetVEMDataByRFID.BeginReqMem := FALSE;
       ELSIF #IO_VIDS.ReplaceTag.BeginReqMem THEN
           #IO_VIDS.ReplaceTag.OkBegin := TRUE;
           #IO_VIDS.ReplaceTag.BeginReqMem := FALSE;
       ELSIF #IO_VIDS.Track.BeginReqMem  THEN
           #IO_VIDS.Track.OkBegin := TRUE;
           #IO_VIDS.Track.BeginReqMem := FALSE;
       ELSIF #IO_VIDS.Confirm.BeginReqMem  THEN
           #IO_VIDS.Confirm.OkBegin := TRUE;
           #IO_VIDS.Confirm.BeginReqMem := FALSE;
       ELSIF #IO_VIDS.Couple.BeginReqMem  THEN
           #IO_VIDS.Couple.OkBegin := TRUE;
           #IO_VIDS.Couple.BeginReqMem := FALSE;
       ELSIF #IO_VIDS.DeCouple.BeginReqMem THEN
           #IO_VIDS.DeCouple.OkBegin := TRUE;
           #IO_VIDS.DeCouple.BeginReqMem := FALSE;
       ELSIF #IO_VIDS.GetNextID.BeginReqMem THEN
           #IO_VIDS.GetNextID.OkBegin := TRUE;
           #IO_VIDS.GetNextID.BeginReqMem := FALSE;
       ELSIF #IO_VIDS.GetSpecData.BeginReqMem  THEN
           #IO_VIDS.GetSpecData.OkBegin := TRUE;
           #IO_VIDS.GetSpecData.BeginReqMem := FALSE;
       ELSIF #IO_VIDS.PutSpecData.BeginReqMem  THEN
           #IO_VIDS.PutSpecData.OkBegin := TRUE;
           #IO_VIDS.PutSpecData.BeginReqMem := FALSE;
       END_IF;

       //Initialize commands
       #CmdCodeSent := 0;
       #CmdCodeRcvd := 0;

       //Initialize
       IF NOT #IO_VIDS.Track.OkBegin  AND NOT #IO_VIDS.GetNextID.OkBegin AND NOT #IO_VIDS.Confirm.OkBegin THEN

           //Initialize IO_VIDS.VEMData
           #DeserializePos := 0;
           #RetVal := Deserialize(SRC_ARRAY := #VEMDataInitArray, DEST_VARIABLE => #IO_VIDS.VEMData, POS := #DeserializePos);
           #RetVal := FILL(BVAL := #SPACE, BLK => #IO_VIDS.VEMData.UserID);
           #RetVal := FILL(BVAL := #SPACE, BLK => #IO_VIDS.VEMData.Variant);
           #RetVal := FILL(BVAL := #SPACE, BLK => #IO_VIDS.VEMData.VinNumber);
           #RetVal := FILL(BVAL := #SPACE, BLK => #IO_VIDS.VEMData.PopIDSuffix);

           //Initialize IO_VIDS.Specific data
           #RetVal := FILL(BVAL := #EmptyByte, BLK => #IO_VIDS.SpecificDataInit);

           //Initialize IO_VEMData
           #DeserializePos := 0;
           #RetVal := Deserialize(SRC_ARRAY := #VEMDataInitArray, DEST_VARIABLE => #IO_VEMData, POS := #DeserializePos);
           #RetVal := FILL(BVAL := #SPACE, BLK => #IO_VEMData.UserID);
           #RetVal := FILL(BVAL := #SPACE, BLK => #IO_VEMData.Variant);
           #RetVal := FILL(BVAL := #SPACE, BLK => #IO_VEMData.VinNumber);
           #RetVal := FILL(BVAL := #SPACE, BLK => #IO_VEMData.PopIDSuffix);

           //Initialize IO_Specific data
           #RetVal := FILL(BVAL := #EmptyByte, BLK => #IO_SpecificData);

           //Reset validation
           #VEMDataValid := FALSE;
           #VEMDataNotValid := FALSE;

       END_IF;

   ELSE
       #IO_VIDS.GetVEMData.OkBegin := FALSE;
       #IO_VIDS.ChangeData.OkBegin := FALSE;
       #IO_VIDS.InitTag.OkBegin := FALSE;
       #IO_VIDS.GetVEMDataByRFID.OkBegin := FALSE;
       #IO_VIDS.ReplaceTag.OkBegin := FALSE;
       #IO_VIDS.Track.OkBegin := FALSE;
       #IO_VIDS.Confirm.OkBegin := FALSE;
       #IO_VIDS.Couple.OkBegin := FALSE;
       #IO_VIDS.DeCouple.OkBegin := FALSE;
       #IO_VIDS.GetNextID.OkBegin := FALSE;
       #IO_VIDS.GetSpecData.OkBegin := FALSE;
       #IO_VIDS.PutSpecData.OkBegin := FALSE;
       #OkBegin := False;

   END_IF;

   //Step 50 on Active - Step Timer - Start
   #_Step50Tmr(I_StartTimer:=#StepNbr=50,
               I_HoldTimer:=FALSE,
               I_MaxTimerValue:=5000,
               O_TimerResult=>#Step50TmrElapsed,
               O_TimerValue=>#Step50TmrAct);

   //Step 50 On Active - Step Timer - Error overtime
   IF #Step50TmrElapsed THEN
       #Status := #STAT_CODE_RCV_NEW_DATA_OVTIME;
   END_IF;

   //Step 50 On Active - Step Timer - Memorize maximum
   IF #Step50TmrAct > #Step50TmrActMax THEN
       #Step50TmrActMax := #Step50TmrAct;
   END_IF;

   (******************************************************************************)
   (* Step 50 TO 100                                                             *)
   (******************************************************************************)

   //Step 50 to 100
   IF #Step50To100Cond THEN
       #StepNbr := 100;
       #Step100EntryPls := TRUE;
   ELSE
       #Step100EntryPls := FALSE;
   END_IF;

   //Step 50 to 200
   IF #Step50To200Cond THEN
       #StepNbr := 200;
       #Step200EntryPls := TRUE;
   ELSE
       #Step200EntryPls := FALSE;
   END_IF;

   //Step 0 - Exit pulse
   #Step0ExitPls := #Step50EntryPls;

   //Step 50 to 100 - Condition
   #Step50To100Cond := #StepNbr = 50 AND #IO_VIDS.GetVEMDataByRFID.Running;

   //Step 50 TO 200 - Condition
   #Step50To200Cond:= #StepNbr=50 AND
   (#IO_VIDS.GetVEMData.Running OR
   #IO_VIDS.ChangeData.Running OR
   #IO_VIDS.InitTag.Running OR
   #IO_VIDS.ReplaceTag.Running OR
   #IO_VIDS.Track.Running OR
   #IO_VIDS.Confirm.Running OR
   #IO_VIDS.Couple.Running OR
   #IO_VIDS.DeCouple.Running OR
   #IO_VIDS.GetNextID.Running OR
   #IO_VIDS.GetSpecData.Running OR
   #IO_VIDS.PutSpecData.Running);

   (******************************************************************************)
   (* Step 100                                                                   *)
   (******************************************************************************)

   // Step 0 On Exit
   IF #Step0ExitPls THEN

       #Status := #STAT_CODE_BUSY; //Status busy

   END_IF;


   //Step 100 On Active - New data received
   IF #StepNbr = 100 AND #NewData THEN
       //Copy received VEM data
       #RetVal := BLKMOV(SRCBLK := #ptrVEMDataVDCommLocalRcv, DSTBLK => #VEMDataRcvArray);
       #DeserializePos := 0;
       #RetVal:=Deserialize(SRC_ARRAY := #VEMDataRcvArray, DEST_VARIABLE => #IO_VIDS.VEMData, POS := #DeserializePos);

       #CmdCodeRcvd := #IO_VIDS.VEMData.CommandCode;
       //Update #Status
       IF #IO_VIDS.VEMData.ErrorCode < 0 THEN
           #Status := DINT_TO_INT(#IO_VIDS.VEMData.ErrorCode);
       ELSE
           #IO_VEMData.Identification := #IO_VIDS.VEMData.Identification;
       END_IF;
   END_IF;

   //Step 100 on Active - Step Timer - Start
   #_Step100Tmr(I_StartTimer := #StepNbr = 100,
                I_HoldTimer := FALSE,
                I_MaxTimerValue := 15000,
                O_TimerResult => #Step100TmrElapsed,
                O_TimerValue => #Step100TmrAct);

   //Step 100 On Active - Step Timer - Error overtime
   IF #Step100TmrElapsed THEN
       #Status := #STAT_CODE_RCV_NEW_DATA_OVTIME;
   END_IF;

   //Step 100 On Active - Step Timer - Memorize maximum
   IF #Step100TmrAct > #Step100TmrActMax THEN
       #Step100TmrActMax := #Step100TmrAct;
   END_IF;

   //Step 100 On EXIT - Store Identification
   IF #Step100ExitPls THEN
       #VD_Identification := #IO_VIDS.VEMData.Identification;
   END_IF;

   (******************************************************************************)
   (* Step 100 to 300                                                            *)
   (******************************************************************************)

   //Step 100 to 300
   IF #Step100To300Cond THEN
       #StepNbr := 300;
       #Step300EntryPls := TRUE;
   ELSE
       #Step300EntryPls := FALSE;
   END_IF;

   //Step 100 to 300 - Condition
   #Step100To300Cond :=
   #StepNbr = 100 AND
   #IO_VIDS.VEMData.CommandCode = 1001 AND
   #Status > 0 AND
   (#IO_VIDS.IDType = 0 AND #IO_VIDS.VEMData.Identification <> 0 OR #IO_VIDS.IDType > 0 AND #IO_VIDS.VEMData.CarrierID <> 0) AND
   NOT #NewData;

   (******************************************************************************)
   (* Step 200 - Send data                                                       *)
   (******************************************************************************)

   //Step 200 - On Entry - Check VEM data
   #DataValidSnd := #Step200EntryPls AND #IO_VIDS.VEMData.CommandCode <> 0;

   //Step 200 - On Entry - Check VEM data - Error
   IF #Step200EntryPls AND NOT #DataValidSnd THEN
       #Status := #STATUS_MINUS_006;
   END_IF;

   //Step 200 On Entry - VDCommLocalSndDB - Send VEM data TO virtual device
   IF #Step200EntryPls AND #Status > 0 THEN
       #SerializePos := 0;
       #RetVal:=Serialize(SRC_VARIABLE:=#IO_VIDS.VEMData, DEST_ARRAY=>#VEMDataSndArray, POS:=#SerializePos);
       #RetVal:=BLKMOV(SRCBLK := #VEMDataSndArray, DSTBLK => #ptrVEMDataVDCommLocalSnd);
       #RetVal:=BLKMOV(SRCBLK := #IO_VIDS.SpecificDataInit, DSTBLK => #ptrSpecDataVDCommLocalSnd);
       #CmdCodeSent := #IO_VIDS.VEMData.CommandCode;
   END_IF;

   //Step 200 on Active - Step Timer - Start
   #_Step200Tmr(I_StartTimer := #StepNbr = 200,
                I_HoldTimer := FALSE,
                I_MaxTimerValue := 15000,
                O_TimerResult => #Step200TmrElapsed,
                O_TimerValue => #Step200TmrAct);

   //Step 200 On Active - Step Timer - Error overtime
   IF #Step200TmrElapsed THEN
       #Status := #STATUS_MINUS_003;
   END_IF;

   //Step 200 On Active - Step Timer - Memorize maximum
   IF #Step200TmrAct > #Step200TmrActMax THEN
       #Step200TmrActMax := #Step200TmrAct;
   END_IF;

   //Step 200 On Active - Send TO VD
   #SendToVD := #StepNbr = 200 AND #Status>0;

   (******************************************************************************)
   (* Step 200 to 300                                                            *)
   (******************************************************************************)

   //Step 200 to 300
   IF #Step200To300Cond THEN
       #StepNbr := 300;
       #Step200ExitPls := TRUE;
   ELSE
       #Step200ExitPls := FALSE;
   END_IF;

   //Step 200 to 300 - Condition
   #Step200To300Cond := #StepNbr = 200 AND #SendFinished AND #Status > 0;

   (******************************************************************************)
   (* Step 300                                                                   *)
   (******************************************************************************)

   //Step 300 On Entry - VDCommLocalRcvDB - Create pointer TO VEM data
   #ptrVEMDataVDCommLocalRcvStruct.ID := #POINTER_SYNTAX_ID;
   #ptrVEMDataVDCommLocalRcvStruct.DataType := #DATA_TYPE_BYTE;
   #ptrVEMDataVDCommLocalRcvStruct.ReplicationFactor := 256;
   #ptrVEMDataVDCommLocalRcvStruct.DbNbr := UINT_TO_WORD(DB_ANY_TO_UINT(#C_VDCommLocalRcvDB));
   #ptrVEMDataVDCommLocalRcvStruct.CrossAreaPointer := SHL(IN := #VDCOM_VEM_DATA_OFFSET, N := 3) OR #AREA_IDENTIFIER; //Offset 10

   //Step 300 On Entry - VDCommLocalRcvDB - Create pointer TO Specific data
   #ptrSpecDataVDCommLocalRcvStruct.ID := #POINTER_SYNTAX_ID;
   #ptrSpecDataVDCommLocalRcvStruct.DataType := #DATA_TYPE_BYTE;
   #ptrSpecDataVDCommLocalRcvStruct.ReplicationFactor := 2048;
   #ptrSpecDataVDCommLocalRcvStruct.DbNbr := UINT_TO_WORD(DB_ANY_TO_UINT(#C_VDCommLocalRcvDB));
   #ptrSpecDataVDCommLocalRcvStruct.CrossAreaPointer := SHL(IN := #VDCOM_SPEC_DATA_OFFSET, N := 3) OR #AREA_IDENTIFIER; //Offset 10

   //Step 300 On Active - Receive data from virtual device
   IF #StepNbr = 300 AND #NewData THEN

       //Copy received data to VEM data receive structure
       #RetVal := BLKMOV(SRCBLK := #ptrVEMDataVDCommLocalRcv, DSTBLK => #VEMDataRcvArray);
       #DeserializePos := 0;
       #RetVal := Deserialize(SRC_ARRAY := #VEMDataRcvArray, DEST_VARIABLE => #VEMDataRcv, POS := #DeserializePos);

       //Received command code
       #CmdCodeRcvd := #VEMDataRcv.CommandCode;

       //Check error code
       IF #VEMDataRcv.ErrorCode < 0 THEN
           #Status := DINT_TO_INT(#VEMDataRcv.ErrorCode);
           //Data not Valid signal
           #VEMDataNotValid := TRUE;
       ELSE
           //Check data
           #DataValidRcv := NOT #IO_VIDS.GetVEMDataByRFID.Running AND
           #VEMDataRcv.CommandCode = #IO_VIDS.VEMData.CommandCode;

           #DataValidRcvGetVEMDataByRFID := #IO_VIDS.GetVEMDataByRFID.Running AND
           ((#VEMDataRcv.IdType = 0 AND #VEMDataRcv.Identification <> 0) OR (#VEMDataRcv.IdType <> 0 AND #VEMDataRcv.CarrierID <> 0));

           IF #DataValidRcv OR #DataValidRcvGetVEMDataByRFID THEN

               //Status 001 : Success
               #Status := #STATUS_001;

               //Copy all data
               #DeserializePos := 0;
               #RetVal := Deserialize(SRC_ARRAY := #VEMDataRcvArray, DEST_VARIABLE => #IO_VIDS.VEMData, POS := #DeserializePos);
               #RetVal := BLKMOV(SRCBLK := #ptrSpecDataVDCommLocalRcv, DSTBLK => #IO_SpecificData);
               #DeserializePos := 0;
               #RetVal := Deserialize(SRC_ARRAY := #VEMDataRcvArray, DEST_VARIABLE => #IO_VEMData, POS := #DeserializePos);
               #DeserializePos := 0;
               #RetVal := Deserialize(SRC_ARRAY := #VEMDataRcvArray, DEST_VARIABLE => #IO_VEMDataChange, POS := #DeserializePos);

               //Data Valid signal
               #VEMDataValid := TRUE;

           ELSE
               #VEMDataNotValid := TRUE;
               #Status := #STATUS_MINUS_005;
           END_IF;
       END_IF;
   END_IF;

   //Step 300 on Active - Step Timer - Start
   #_Step300Tmr(I_StartTimer := #StepNbr = 300,
                I_HoldTimer := FALSE,
                I_MaxTimerValue := 15000,
                O_TimerResult => #Step300TmrElapsed,
                O_TimerValue => #Step300TmrAct);

   //Step 300 On Active - Step Timer - Error overtime
   IF #Step300TmrElapsed THEN
       #Status := #STATUS_MINUS_009;
   END_IF;

   //Step 300 On Active - Step Timer - Memorize maximum
   IF #Step300TmrAct > #Step300TmrActMax THEN
       #Step300TmrActMax := #Step300TmrAct;
   END_IF;

   (******************************************************************************)
   (* Step 300 to 400                                                            *)
   (******************************************************************************)

   //Step 300 to 400
   IF #Step300To400Cond THEN
       #StepNbr := 400;
       #Step300ExitPls := TRUE;
   ELSE
       #Step300ExitPls := FALSE;
   END_IF;

   //Step 300 TO 400 - Condition
   #Step300To400Cond := #StepNbr = 300 AND #Status = 1;

   (******************************************************************************)
   (* Step XXX to 400                                                            *)
   (******************************************************************************)

   //Step XXX TO 400
   IF #StepNbr > 0 AND #Status < 0 THEN
       #VEMDataNotValid := TRUE;
       #StepNbr := 400;
   END_IF;

   (******************************************************************************)
   (* Step 400 to 0                                                              *)
   (******************************************************************************)

   //Step 400 to 0
   IF #Step400To0Cond THEN
       #StepNbr := 0;
       #Step400ExitPls := TRUE;
   ELSE
       #Step400ExitPls := FALSE;
   END_IF;

   //Step 400 TO 0 - Condition
   #Step400To0Cond := #StepNbr = 400;

   (******************************************************************************)
   (* Step 400 - Finish & Final Status                                           *)
   (******************************************************************************)

   //Step 400 On active - Finish & Final Status
   IF #StepNbr = 400 THEN

       IF #IO_VIDS.GetVEMData.Running THEN
           #IO_VIDS.GetVEMData.Running := FALSE;
           #IO_VIDS.GetVEMData.Status := #Status;
           #IO_VIDS.GetVEMData.Finished := TRUE;
       ELSIF #IO_VIDS.ChangeData.Running THEN
           #IO_VIDS.ChangeData.Running := FALSE;
           #IO_VIDS.ChangeData.Status := #Status;
           #IO_VIDS.ChangeData.Finished := TRUE;
       ELSIF #IO_VIDS.InitTag.Running THEN
           #IO_VIDS.InitTag.Running := FALSE;
           #IO_VIDS.InitTag.Status := #Status;
           #IO_VIDS.InitTag.Finished := TRUE;
       ELSIF #IO_VIDS.GetVEMDataByRFID.Running THEN
           #IO_VIDS.GetVEMDataByRFID.Running := FALSE;
           #IO_VIDS.GetVEMDataByRFID.Status := #Status;
           #IO_VIDS.GetVEMDataByRFID.Finished := TRUE;
       ELSIF #IO_VIDS.ReplaceTag.Running THEN
           #IO_VIDS.ReplaceTag.Running := FALSE;
           #IO_VIDS.ReplaceTag.Status := #Status;
           #IO_VIDS.ReplaceTag.Finished := TRUE;
       ELSIF #IO_VIDS.Track.Running THEN
           #IO_VIDS.Track.Running := FALSE;
           #IO_VIDS.Track.Status := #Status;
           #IO_VIDS.Track.Finished := TRUE;
       ELSIF #IO_VIDS.Confirm.Running THEN
           #IO_VIDS.Confirm.Running := FALSE;
           #IO_VIDS.Confirm.Status := #Status;
           #IO_VIDS.Confirm.Finished := TRUE;
       ELSIF #IO_VIDS.Couple.Running THEN
           #IO_VIDS.Couple.Running := FALSE;
           #IO_VIDS.Couple.Status := #Status;
           #IO_VIDS.Couple.Finished := TRUE;
       ELSIF #IO_VIDS.DeCouple.Running THEN
           #IO_VIDS.DeCouple.Running := FALSE;
           #IO_VIDS.DeCouple.Status := #Status;
           #IO_VIDS.DeCouple.Finished := TRUE;
       ELSIF #IO_VIDS.GetNextID.Running THEN
           #IO_VIDS.GetNextID.Running := FALSE;
           #IO_VIDS.GetNextID.Status := #Status;
           #IO_VIDS.GetNextID.Finished := TRUE;
       ELSIF #IO_VIDS.GetSpecData.Running THEN
           #IO_VIDS.GetSpecData.Running := FALSE;
           #IO_VIDS.GetSpecData.Status := #Status;
           #IO_VIDS.GetSpecData.Finished := TRUE;
       ELSIF #IO_VIDS.PutSpecData.Running THEN
           #IO_VIDS.PutSpecData.Running := FALSE;
           #IO_VIDS.PutSpecData.Status := #Status;
           #IO_VIDS.PutSpecData.Finished := TRUE;
       END_IF;

   ELSE

       #IO_VIDS.GetVEMData.Finished := FALSE;
       #IO_VIDS.ChangeData.Finished := FALSE;
       #IO_VIDS.InitTag.Finished := FALSE;
       #IO_VIDS.GetVEMDataByRFID.Finished := FALSE;
       #IO_VIDS.ReplaceTag.Finished := FALSE;
       #IO_VIDS.Track.Finished := FALSE;
       #IO_VIDS.Confirm.Finished := FALSE;
       #IO_VIDS.Couple.Finished := FALSE;
       #IO_VIDS.DeCouple.Finished := FALSE;
       #IO_VIDS.GetNextID.Finished := FALSE;
       #IO_VIDS.GetSpecData.Finished := FALSE;
       #IO_VIDS.PutSpecData.Finished := FALSE;

   END_IF;

   (******************************************************************************)
   (* CPU1500 - VDComSubSystem                                                   *)
   (******************************************************************************)

   //Reset NewData
   #ResetNewData:=#NewData;

   #MessageLength := DWORD_TO_WORD(#IO_VIDS.VEMData.SpecificDataLength+266);

   #"_LVDComSubSystemS7-1500"(I_CommunicationReset:=#ResetAllRequests,
                              I_SendRequest:=#SendToVD,
                              I_ResetNewData:=#ResetNewData,
                              I_MasterNewMessage:=#IO_VDComm.NewMessageVD,
                              I_MasterSendFinished:=#IO_VDComm.MessageSendDoneVD,
                              I_VDCommRecvDB:=#C_VDCommMasterRcvDB,
                              I_VDCommSendDB:=#C_VDCommMasterSndDB,
                              C_LocalRecvDB:=#C_VDCommLocalRcvDB,
                              C_LocalSendDB:=#C_VDCommLocalSndDB,
                              C_MessType:=20562,
                              C_SubSystem:=#C_SubSystem,
                              C_SendMessLen:=#MessageLength,
                              O_SendFinished=>#SendFinished,
                              O_NewData=>#NewData,
                              IO_MasterSendReq:=#IO_VDComm.MasterSendReq,
                              IO_MasterAckReq:=#IO_VDComm.MasterAckReq,
                              IO_SubSystemDBNr:=#IO_VDComm.VDCommSendDBNr,
                              IO_VDCommSendDB:=#IO_VDComm.VDCommSendDB);


   (******************************************************************************)
   (* Common signals to all submodules                                           *)
   (******************************************************************************)

   //Common signals to all submodules
   #IO_VIDS.PartPres := #PartPres;
   #IO_VIDS.IDType := #C_IDType;
   #IO_VIDS.VEMDataValid := #VEMDataValid;
   #IO_VIDS.VEMDataNotValid := #VEMDataNotValid;
   #IO_VIDS.CmdCodeRcvd := #CmdCodeRcvd;
   #IO_VIDS.CmdCodeSent := #CmdCodeSent;

   (******************************************************************************)
   (* Outputs                                                                    *)
   (******************************************************************************)

   IF #SECTION_OUTPUTS THEN

       #O_GetVEMDataBusy := #BusyGetVEMData;
       #O_Status := #Status;
       #O_Alarm := #Status < 0;
       #O_VEMDataValid := #VEMDataValid;
       #O_VEMDataNotValid := #VEMDataNotValid;

   END_IF;

   (******************************************************************************)
   (* HMI                                                                        *)
   (******************************************************************************)

   IF #SECTION_HMI THEN

       //Decode - BodyType matrix - Car type
       #CarTypeBody := DINT_TO_INT(DWORD_TO_DINT(#IO_VEMData.BodyTypeMatrix) / 100000);

       //Decode - BodyType matrix - Steering
       #SteeringBody := DINT_TO_INT((DWORD_TO_DINT(#IO_VEMData.BodyTypeMatrix) / 100000) MOD 10);

       //Decode - Variant - Car type - First digit
       #CarTypeArray[1] := (CHAR_TO_INT(#IO_VEMData.Variant[1]) - 48) * 100;
       #CarTypeArray[2] := (CHAR_TO_INT(#IO_VEMData.Variant[2]) - 48) * 10;
       #CarTypeArray[3] := (CHAR_TO_INT(#IO_VEMData.Variant[3]) - 48);

       //Decode - Variant - Car type - Summary digits
       #CarTypeVariant := #CarTypeArray[1] + #CarTypeArray[2] + #CarTypeArray[3];

       //Decode - Variant - Steering
       #SteeringVariant := #IO_VEMData.Variant[10];

       //HMI - Message - Part Present - Visible
       IF #IO_VIDS.PartPres THEN
           #H_Master.H_msgPartPresAnim := #VISIBLE;
       ELSE
           #H_Master.H_msgPartPresAnim := #OFF;
       END_IF;

       //HMI - Message - VEM Data Valid - Visible
       IF #VEMDataValid THEN
           #H_Master.H_msgVEMDataValidAnim := #VISIBLE;
       ELSE
           #H_Master.H_msgVEMDataValidAnim := #OFF;
       END_IF;

       //HMI - Message - VEM Data not Valid - Visible
       IF #VEMDataNotValid THEN
           #H_Master.H_msgVEMDataNotValidAnim := #VISIBLE;
       ELSE
           #H_Master.H_msgVEMDataNotValidAnim := #OFF;
       END_IF;

       //HMI - Value - Command code sent
       #H_Master.H_txtCommandCodeSent := #CmdCodeSent;

       //HMI - Value - Command code received
       #H_Master.H_txtCommandCodeRcvd := #CmdCodeRcvd;

       (******************************************************************************)
       (* HMI - Vehicle types                                                        *)
       (******************************************************************************)

       //HMI - Message - Body VEM data
       IF #C_IDType = 0 THEN
           #H_Master.H_msgVEMDataBody := 1;
       ELSE
           #H_Master.H_msgVEMDataBody := 0;
       END_IF;

       //HMI - Message - Carrier VEM data
       IF #C_IDType = 0 THEN
           #H_Master.H_msgVEMDataCarrier := 1;
       ELSE
           #H_Master.H_msgVEMDataCarrier := 0;
       END_IF;

       #H_Master.H_txtIdentification := #IO_VEMData.Identification;                    //HMI - Value - TagID
       #H_Master.H_txtBodyID := #IO_VEMData.BodyID;                                    //HMI - Value - BodyID
       #H_Master.H_txtCarrierID := #IO_VEMData.CarrierID;                              //HMI - Value - CarrierID
       #H_Master.H_txtBodyTypeMatrix := #IO_VEMData.BodyTypeMatrix;                    //HMI - Value - Bodytype matrix
       #H_Master.H_txtRouting := #IO_VEMData.Routing;                                  //HMI - Value - Routing
       #H_Master.H_txtCarrierDestination := #IO_VEMData.Destination;                   //HMI - Value - Carrier Destination
       #H_Master.H_txtWorkUntil := #IO_VEMData.WorkUntil;                              //HMI - Value - Work UNTIL Station
       #H_Master.H_txtWorkAfter := #IO_VEMData.BegWorkAfter;                           //HMI - Value - Start Work After Station
       #H_Master.H_txtBodyCargoStatus := #IO_VEMData.BodyCargoStatus ;                 //HMI - Value - Body Cargo Status
       #H_Master.H_txtCarrierCargoStatus := #IO_VEMData.CarrierCargoStatus;            //HMI - Value - Carrier Cargo Status
       #H_Master.H_txtEquipmentWork := #IO_VEMData.EquipmentWork;                      //HMI - Value - Equipment Work
       #H_Master.H_txtAvailabilityStatus := #IO_VEMData.AvailabilityStatus;            //HMI - Value - Availability Status
       #H_Master.H_txtModelYear := #IO_VEMData.ModelYear;                              //HMI - Value - ModelYear
       #H_Master.H_txtPreSerieInfo := #IO_VEMData.PreSerieInfo;                        //HMI - Value - Preseries Info
       #H_Master.H_txtWorkStatus := #IO_VEMData.WorkStatus;                            //HMI - Value - Work Status
       #H_Master.H_txtBodyType1 := #IO_VEMData.BodyType1;                              //HMI - Value - Bodytype 1
       #H_Master.H_txtBodyType2 := #IO_VEMData.BodyType2;                              //HMI - Value - Bodytype 2
       #H_Master.H_txtRobotProgramNumber := #IO_VEMData.RobotProgramNumber;            //HMI - Value - Robot Program Number
       #H_Master.H_txtPLCProgramNbr := #H_Master.H_txtPLCProgramNbr;                   //HMI - Value - PLC Program Number
       #H_Master.H_txtEquipmentWorkDone := #IO_VEMData.EquipmentWorkDone;              //HMI - Value - Equipment Work Done
       #H_Master.H_txtSequenceNumber := #IO_VEMData.SequenceNumber;                    //HMI - Value - Sequence Number
       #H_Master.H_txtBufferIn := #IO_VEMData.BufferIn;                                //HMI - Value - BufferIn
       #H_Master.H_txtBufferOut := #IO_VEMData.BufferOut;                              //HMI - Value - BufferOut
       #H_Master.H_txtCarrierType := #IO_VEMData.CarrierType;                          //HMI - Value - Carrier Type
       #H_Master.H_txtCarrierLapCounter := #IO_VEMData.CarrierLapCounter;              //HMI - Value - Carrier Lap Counter
       #H_Master.H_txtCarrierIDUBFlow := #IO_VEMData.CarrierIDUBFlow;                  //HMI - Value - Carrier ID UB Flow
       #H_Master.H_txtCarrierBodyType := #IO_VEMData.CarrierBodyType;                  //HMI - Value - Carrier Bodytype
       #H_Master.H_txtAddQualityItemEquipment := #IO_VEMData.AddQualityItemEquipment;  //HMI - Value - Add Quality Item Equipment
       #H_Master.H_txtChkQualityItemEquipment := #IO_VEMData.CheckQualityItemEquipment;//HMI - Value - Check Quality Item Equipment
       #H_Master.H_txtCarrierMaxCycleCounter := #IO_VEMData.CarrierMaxCycleCount;      //HMI - Value - CarrMaxCycleCntr    
       #H_Master.H_txtSurfacerColour := #IO_VEMData.SurfacerColour;                    //HMI - Value - SurfacerColour
       #H_Master.H_txtTopCoatColour := #IO_VEMData.TopCoatColour;                      //HMI - Value - TopCoatColour
       #H_Master.H_txtClearCoatColour := #IO_VEMData.ClearCoatColour;                  //HMI - Value - ClearCoatColour
       #H_Master.H_txtPopType := #IO_VEMData.PopType;                                  //HMI - Value - PopType
       #H_Master.H_txtPopId := #IO_VEMData.PopID;                                      //HMI - Value - PopId
       #H_Master.H_txtPopIdSuffix := #IO_VEMData.PopIDSuffix;                          //HMI - Value - PopId

       //HMI - Value - Variant
       FOR #i := 1 TO 8 DO
           #H_Master.H_txtVariant[#i] := #IO_VEMData.Variant[#i];
       END_FOR;

       //HMI - Value - VIN number
       FOR #i := 1 TO 20 DO
           #H_Master.H_txtVinNumber[#i - 1] := #IO_VEMData.VinNumber[#i];
       END_FOR;

       #H_Master.H_txtMixNumber := #IO_VEMData.MixNumber;                          //HMI - Value - Mixnumber
       #H_Master.H_txtIDType := #IO_VEMData.IdType;                                // HMI - Value - ID Type

       //HMI - Message - Running 
       #H_Master.H_msgFunctionNbrAnim := 0;                //Reset animation before we begin

       //HMI - Message - Running - Get VEM Data
       IF #IO_VIDS.GetVEMData.Running THEN
           #H_Master.H_msgFunctionNbrAnim := 1;
       END_IF;

       //HMI - Message - Running - Change VEM Data
       IF #IO_VIDS.ChangeData.Running THEN
           #H_Master.H_msgFunctionNbrAnim := 2;
       END_IF;

       //HMI - Message - Running - Init
       IF #IO_VIDS.InitTag.Running THEN
           #H_Master.H_msgFunctionNbrAnim := 3;
       END_IF;

       //HMI - Message - Running - Get VEM Data by RFID
       IF #IO_VIDS.GetVEMDataByRFID.Running THEN
           #H_Master.H_msgFunctionNbrAnim := 4;
       END_IF;

       //HMI - Message - Running - Replace tag
       IF #IO_VIDS.ReplaceTag.Running THEN
           #H_Master.H_msgFunctionNbrAnim := 5;
       END_IF;

       //HMI - Message - Running - Track
       IF #IO_VIDS.Track.Running THEN
           #H_Master.H_msgFunctionNbrAnim := 6;
       END_IF;

       //HMI - Message - Running - Confirm
       IF #IO_VIDS.Confirm.Running THEN
           #H_Master.H_msgFunctionNbrAnim := 7;
       END_IF;

       //HMI - Message - Running - Couple
       IF #IO_VIDS.Couple.Running THEN
           #H_Master.H_msgFunctionNbrAnim := 8;
       END_IF;

       //HMI - Message - Running - Decouple
       IF #IO_VIDS.DeCouple.Running THEN
           #H_Master.H_msgFunctionNbrAnim := 9;
       END_IF;

       //HMI - Message - Running - Get Next ID
       IF #IO_VIDS.GetNextID.Running THEN
           #H_Master.H_msgFunctionNbrAnim := 10;
       END_IF;

       //HMI - Message - Running - Get Specific Data
       IF #IO_VIDS.GetSpecData.Running THEN
           #H_Master.H_msgFunctionNbrAnim := 11;
       END_IF;

       //HMI - Message - Running - Put Specific Data
       IF #IO_VIDS.PutSpecData.Running THEN
           #H_Master.H_msgFunctionNbrAnim := 12;
       END_IF;

       #H_Master.H_msgStepNbrAnim := INT_TO_WORD(#StepNbr);             //HMI - Message - StepNumber

       //Update step timers
       IF #StepNbr = 100 THEN
           #H_Master.H_txtStep100TmrMax := DINT_TO_INT(#Step100TmrAct);  //HMI - Step 100 Timer
       ELSIF #StepNbr = 200 THEN
           #H_Master.H_txtStep200TmrMax := DINT_TO_INT(#Step200TmrAct);  //HMI - Step 200 Timer
       ELSIF #StepNbr = 300 THEN
           #H_Master.H_txtStep300TmrMax := DINT_TO_INT(#Step300TmrAct);  //HMI - Step 300 Timer
       END_IF;

       //Reset Step timers
       IF #H_Master.H_btnResetStepTimers <> 0 THEN
           #H_Master.H_txtStep100TmrMax := 0;
           #H_Master.H_txtStep200TmrMax := 0;
           #H_Master.H_txtStep300TmrMax := 0;
       END_IF;

       #H_Master.H_msgStatus := #Status;                   //HMI - Status

       // HMI - Icon animation
       "LIAnimDWord"(I_SetPos := FALSE,
                     I_ResetPos := FALSE,
                     I_Active := #Status > 1,
                     I_Visible := FALSE,
                     I_OutOfUse := FALSE,
                     I_IntlkSet := FALSE,
                     I_IntlkReset := FALSE,
                     I_IntlkSetAlm := FALSE,
                     I_IntlkResetAlm := FALSE,
                     I_ManualMode := FALSE,
                     I_FncSelInHMI := FALSE,
                     I_AnySelected := FALSE,
                     I_AlarmA := FALSE,
                     I_AlarmB := FALSE,
                     I_AlarmC := #Status < 0,
                     I_AlarmD := FALSE,
                     I_SafetyOk := FALSE,
                     I_Service:="TRUE",
                     I_Spare1:="FALSE",
                     I_Spare2:="FALSE",
                     I_Spare3:="FALSE",
                     I_Spare4:="FALSE",
                     I_Spare5:="FALSE",
                     I_Spare6:="FALSE",
                     I_Spare7:="FALSE",
                     I_Spare8:="FALSE",
                     I_Spare9:="FALSE",
                     I_Spare10:="FALSE",
                     I_Spare11:="FALSE",
                     I_Spare12:="FALSE",
                     I_Spare13:="FALSE",
                     I_Spare14:="FALSE",
                     H_IAnim => #H_HMI.H_IAnim);

   (******************************************************************************)
   (* HMI - Reset buttons                                                        *)
   (******************************************************************************)

       #H_Master.H_btnResetStepTimers := #OFF;
       #H_Master.H_btnGetVEMDataByTagID := #OFF;
       #H_Master.H_btnGetVEMDataByBodyID := #OFF;
       #H_Master.H_btnGetVEMDataByCarrierID := #OFF;
       #H_Master.H_btnGetVEMDataByMixNbr := #OFF;

   END_IF;

   (******************************************************************************)
   (* Alarm                                                                      *)
   (******************************************************************************)

   #Alarm := (#Status < 0);

   "LAlarmSummary"(I_AlarmA := "FALSE",
                   I_AlarmB := "FALSE",
                   I_AlarmC := #Alarm,
                   I_AlarmD := "FALSE",
                   I_AlarmABCondition := "FALSE",
                   IO_Alarm := #IO_Alarm,
                   C_UpperLevelHW := "FALSE",
                   C_UpperLevelSafety := "FALSE",
                   C_Safety := "FALSE",
                   C_Mechanic := "FALSE",
                   C_Transport := "FALSE",
                   C_Feature1 := "FALSE",
                   C_Feature2 := "FALSE",
                   C_Feature3 := "FALSE");
END_FUNCTION_BLOCK
